{attribute 'GeneratedUsingTerminal: EM7004-0000-0017'}
{attribute addProperty BoxType "EM7004-0000-0017"}
{attribute addProperty Id "ControlAT %Q*Control_F189B7373Set_counter_valueAT %Q*UINT2"}
{attribute addProperty CRC "780319811"}
{attribute addProperty Size "5"}
TYPE ENC_Outputs_Channel_2E82BC43 :
STRUCT
	{attribute addProperty Name "Control"}
	Control AT %Q* : Control_F189B737;
	{attribute addProperty Name "Set_counter_value"}
	Set_counter_value AT %Q* : UINT;
END_STRUCT
END_TYPE

(* stored: Version 1.2.0.0, ProductVersion 3.1.4024.9
   DUT ENC_Outputs_Channel_2E82BC43: Id {e5bf8616-6dad-4d7d-ba94-bd477a59f71c} *)
